// TIA Portal V19 export
ORGANIZATION_BLOCK "Main"   // OB1, LAD, ProgramCycle
TITLE = "Main Program Sweep (Cycle)"
{ S7_Optimized_Access := 'TRUE' }
// stored: SetENOAutomatically false
   VAR_INPUT
      Initial_Call : Bool;   // Initial call of this OB
      Remanence : Bool;   // =True, if remanent data are available
   END_VAR
BEGIN

REGION Network 1: Commande reset general
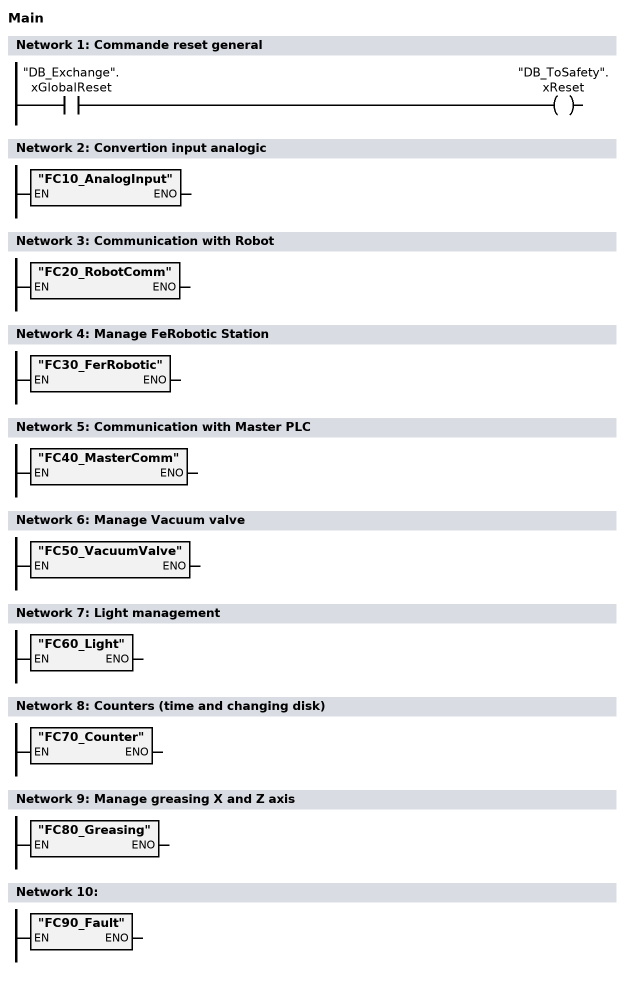
   RUNG wire#powerrail
      Contact( "DB_Exchange".xGlobalReset )
      Coil( "DB_ToSafety".xReset )
   END_RUNG
   // the same network as SCL:
   "DB_ToSafety".xReset := "DB_Exchange".xGlobalReset;
END_REGION

REGION Network 2: Convertion input analogic
   RUNG wire#powerrail
      "FC10_AnalogInput"()
   END_RUNG
   // the same network as SCL:
   "FC10_AnalogInput"();
END_REGION

REGION Network 3: Communication with Robot
   RUNG wire#powerrail
      "FC20_RobotComm"()
   END_RUNG
   // the same network as SCL:
   "FC20_RobotComm"();
END_REGION

REGION Network 4: Manage FeRobotic Station
   RUNG wire#powerrail
      "FC30_FerRobotic"()
   END_RUNG
   // the same network as SCL:
   "FC30_FerRobotic"();
END_REGION

REGION Network 5: Communication with Master PLC
   RUNG wire#powerrail
      "FC40_MasterComm"()
   END_RUNG
   // the same network as SCL:
   "FC40_MasterComm"();
END_REGION

REGION Network 6: Manage Vacuum valve
   RUNG wire#powerrail
      "FC50_VacuumValve"()
   END_RUNG
   // the same network as SCL:
   "FC50_VacuumValve"();
END_REGION

REGION Network 7: Light management
   RUNG wire#powerrail
      "FC60_Light"()
   END_RUNG
   // the same network as SCL:
   "FC60_Light"();
END_REGION

REGION Network 8: Counters (time and changing disk)
   RUNG wire#powerrail
      "FC70_Counter"()
   END_RUNG
   // the same network as SCL:
   "FC70_Counter"();
END_REGION

REGION Network 9: Manage greasing X and Z axis
   RUNG wire#powerrail
      "FC80_Greasing"()
   END_RUNG
   // the same network as SCL:
   "FC80_Greasing"();
END_REGION

REGION Network 10
   RUNG wire#powerrail
      "FC90_Fault"()
   END_RUNG
   // the same network as SCL:
   "FC90_Fault"();
END_REGION
END_ORGANIZATION_BLOCK
